PROGRAM PRG_IM1K4_XTES
VAR
    {attribute 'pytmc' := '
        pv: IM1K4:XTES
        io: io
    '}
    {attribute 'TcLinkTo' := '.bZoomEndFwd := TIIB[IM1K4-EL1088-E5]^Channel 1^Input;
                              .bZoomEndBwd := TIIB[IM1K4-EL1088-E5]^Channel 2^Input;
                              .bFocusEndFwd := TIIB[IM1K4-EL1088-E5]^Channel 3^Input;
                              .bFocusEndBwd := TIIB[IM1K4-EL1088-E5]^Channel 4^Input;
                              .fbOpal.bOpalPower := TIIB[IM1K4-EL2004-E2]^Channel 2^Output;
                              .fbLED.bLedPower := TIIB[IM1K4-EL2004-E2]^Channel 3^Output'}
    fbIM1K4: FB_XPIM;
    {attribute 'TcLinkTo' := '.Status := TIIB[IM1K4-EL6002-E6]^COM TxPDO-Map Inputs Channel 1^Status;
                              .D[0] := TIIB[IM1K4-EL6002-E6]^COM TxPDO-Map Inputs Channel 1^Data In 0;
                              .D[1] := TIIB[IM1K4-EL6002-E6]^COM TxPDO-Map Inputs Channel 1^Data In 1;
                              .D[2] := TIIB[IM1K4-EL6002-E6]^COM TxPDO-Map Inputs Channel 1^Data In 2;
                              .D[3] := TIIB[IM1K4-EL6002-E6]^COM TxPDO-Map Inputs Channel 1^Data In 3;
                              .D[4] := TIIB[IM1K4-EL6002-E6]^COM TxPDO-Map Inputs Channel 1^Data In 4;
                              .D[5] := TIIB[IM1K4-EL6002-E6]^COM TxPDO-Map Inputs Channel 1^Data In 5;
                              .D[6] := TIIB[IM1K4-EL6002-E6]^COM TxPDO-Map Inputs Channel 1^Data In 6;
                              .D[7] := TIIB[IM1K4-EL6002-E6]^COM TxPDO-Map Inputs Channel 1^Data In 7;
                              .D[8] := TIIB[IM1K4-EL6002-E6]^COM TxPDO-Map Inputs Channel 1^Data In 8;
                              .D[9] := TIIB[IM1K4-EL6002-E6]^COM TxPDO-Map Inputs Channel 1^Data In 9;
                              .D[10] := TIIB[IM1K4-EL6002-E6]^COM TxPDO-Map Inputs Channel 1^Data In 10;
                              .D[11] := TIIB[IM1K4-EL6002-E6]^COM TxPDO-Map Inputs Channel 1^Data In 11;
                              .D[12] := TIIB[IM1K4-EL6002-E6]^COM TxPDO-Map Inputs Channel 1^Data In 12;
                              .D[13] := TIIB[IM1K4-EL6002-E6]^COM TxPDO-Map Inputs Channel 1^Data In 13;
                              .D[14] := TIIB[IM1K4-EL6002-E6]^COM TxPDO-Map Inputs Channel 1^Data In 14;
                              .D[15] := TIIB[IM1K4-EL6002-E6]^COM TxPDO-Map Inputs Channel 1^Data In 15;
                              .D[16] := TIIB[IM1K4-EL6002-E6]^COM TxPDO-Map Inputs Channel 1^Data In 16;
                              .D[17] := TIIB[IM1K4-EL6002-E6]^COM TxPDO-Map Inputs Channel 1^Data In 17;
                              .D[18] := TIIB[IM1K4-EL6002-E6]^COM TxPDO-Map Inputs Channel 1^Data In 18;
                              .D[19] := TIIB[IM1K4-EL6002-E6]^COM TxPDO-Map Inputs Channel 1^Data In 19;
                              .D[20] := TIIB[IM1K4-EL6002-E6]^COM TxPDO-Map Inputs Channel 1^Data In 20;
                              .D[21] := TIIB[IM1K4-EL6002-E6]^COM TxPDO-Map Inputs Channel 1^Data In 21'}
    stEL6In AT %I*: EL6InData22b;
    {attribute 'TcLinkTo' := '.Ctrl := TIIB[IM1K4-EL6002-E6]^COM RxPDO-Map Outputs Channel 1^Ctrl;
                              .D[0] := TIIB[IM1K4-EL6002-E6]^COM RxPDO-Map Outputs Channel 1^Data Out 0;
                              .D[1] := TIIB[IM1K4-EL6002-E6]^COM RxPDO-Map Outputs Channel 1^Data Out 1;
                              .D[2] := TIIB[IM1K4-EL6002-E6]^COM RxPDO-Map Outputs Channel 1^Data Out 2;
                              .D[3] := TIIB[IM1K4-EL6002-E6]^COM RxPDO-Map Outputs Channel 1^Data Out 3;
                              .D[4] := TIIB[IM1K4-EL6002-E6]^COM RxPDO-Map Outputs Channel 1^Data Out 4;
                              .D[5] := TIIB[IM1K4-EL6002-E6]^COM RxPDO-Map Outputs Channel 1^Data Out 5;
                              .D[6] := TIIB[IM1K4-EL6002-E6]^COM RxPDO-Map Outputs Channel 1^Data Out 6;
                              .D[7] := TIIB[IM1K4-EL6002-E6]^COM RxPDO-Map Outputs Channel 1^Data Out 7;
                              .D[8] := TIIB[IM1K4-EL6002-E6]^COM RxPDO-Map Outputs Channel 1^Data Out 8;
                              .D[9] := TIIB[IM1K4-EL6002-E6]^COM RxPDO-Map Outputs Channel 1^Data Out 9;
                              .D[10] := TIIB[IM1K4-EL6002-E6]^COM RxPDO-Map Outputs Channel 1^Data Out 10;
                              .D[11] := TIIB[IM1K4-EL6002-E6]^COM RxPDO-Map Outputs Channel 1^Data Out 11;
                              .D[12] := TIIB[IM1K4-EL6002-E6]^COM RxPDO-Map Outputs Channel 1^Data Out 12;
                              .D[13] := TIIB[IM1K4-EL6002-E6]^COM RxPDO-Map Outputs Channel 1^Data Out 13;
                              .D[14] := TIIB[IM1K4-EL6002-E6]^COM RxPDO-Map Outputs Channel 1^Data Out 14;
                              .D[15] := TIIB[IM1K4-EL6002-E6]^COM RxPDO-Map Outputs Channel 1^Data Out 15;
                              .D[16] := TIIB[IM1K4-EL6002-E6]^COM RxPDO-Map Outputs Channel 1^Data Out 16;
                              .D[17] := TIIB[IM1K4-EL6002-E6]^COM RxPDO-Map Outputs Channel 1^Data Out 17;
                              .D[18] := TIIB[IM1K4-EL6002-E6]^COM RxPDO-Map Outputs Channel 1^Data Out 18;
                              .D[19] := TIIB[IM1K4-EL6002-E6]^COM RxPDO-Map Outputs Channel 1^Data Out 19;
                              .D[20] := TIIB[IM1K4-EL6002-E6]^COM RxPDO-Map Outputs Channel 1^Data Out 20;
                              .D[21] := TIIB[IM1K4-EL6002-E6]^COM RxPDO-Map Outputs Channel 1^Data Out 21'}
    stEL6Out AT %Q*: EL6OutData22b;
END_VAR

fbIM1K4.nTransitionAssertionID := 16#2140;
fbIM1K4.nUnknownAssertionID := 16#2149;

fbIM1K4.stOut.fPosition := 0;
fbIM1K4.stOut.bUseRawCounts := FALSE;
fbIM1K4.stOut.nRequestAssertionID := 16#2141;
fbIM1K4.stOut.stBeamParams := PMPS_GVL.cstFullBeam;
fbIM1K4.stOut.bValid := TRUE;

fbIM1K4.stYag.fPosition := -88.87;
fbIM1K4.stYag.bUseRawCounts := FALSE;
fbIM1K4.stYag.nRequestAssertionID := 16#2142;
fbIM1K4.stYag.stBeamParams := PMPS_GVL.cstFullBeam;
fbIM1K4.stYag.bValid := TRUE;

fbIM1K4.stDiamond.fPosition := -58.87;
fbIM1K4.stDiamond.bUseRawCounts := FALSE;
fbIM1K4.stDiamond.nRequestAssertionID := 16#2143;
fbIM1K4.stDiamond.stBeamParams := PMPS_GVL.cstFullBeam;
fbIM1K4.stDiamond.bValid := TRUE;

fbIM1K4.stReticle.fPosition := -28.87;
fbIM1K4.stReticle.bUseRawCounts := FALSE;
fbIM1K4.stReticle.nRequestAssertionID := 16#2144;
fbIM1K4.stReticle.stBeamParams := PMPS_GVL.cst0RateBeam;
fbIM1K4.stReticle.bValid := TRUE;

fbIM1K4(
    fbArbiter := fbArbiter,
    fbFFHWO := fbFastFaultOutput1,
    stYStage := Main.M6,
    stZoomStage := Main.M7,
    stFocusStage := Main.M8,
    stEl6In := stEL6In,
    stEl6Out := stEl6Out);

END_PROGRAM

(* stored: Version 1.1.0.1, ProductVersion 3.1.4022.18
   POU PRG_IM1K4_XTES: Id {7c144f06-c35b-43dd-8fb5-524985d03342}, SpecialFunc None *)
